// Mitsubishi GX Works2 project: 최예현_servo_exam   PLC: Q02/Q02H

PROGRAM MAIN
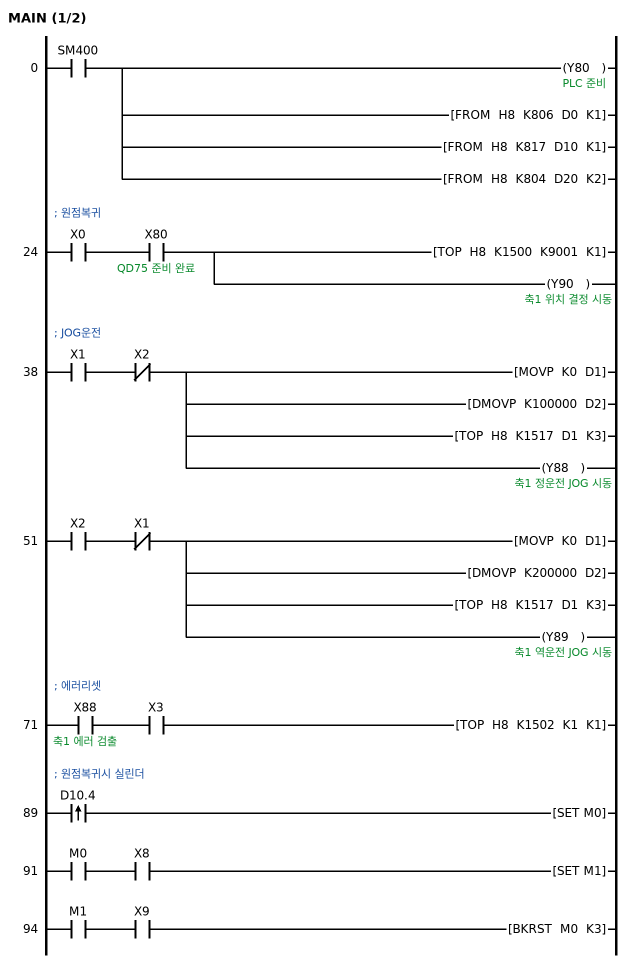
0     LD      SM400
      OUT     Y80  ; PLC 준비
      FROM    H8 K806 D0 K1
      FROM    H8 K817 D10 K1
      FROM    H8 K804 D20 K2
; 원점복귀
24    LD      X0
      AND     X80  ; QD75 준비 완료
      TOP     H8 K1500 K9001 K1
      OUT     Y90  ; 축1 위치 결정 시동
; JOG운전
38    LD      X1
      ANI     X2
      MOVP    K0 D1
      DMOVP   K100000 D2
      TOP     H8 K1517 D1 K3
      OUT     Y88  ; 축1 정운전 JOG 시동
51    LD      X2
      ANI     X1
      MOVP    K0 D1
      DMOVP   K200000 D2
      TOP     H8 K1517 D1 K3
      OUT     Y89  ; 축1 역운전 JOG 시동
; 에러리셋
71    LD      X88  ; 축1 에러 검출
      AND     X3
      TOP     H8 K1502 K1 K1
; 원점복귀시 실린더
89    LDP     D10.4
      SET     M0
91    LD      M0
      AND     X8
      SET     M1
94    LD      M1
      AND     X9
      BKRST   M0 K3
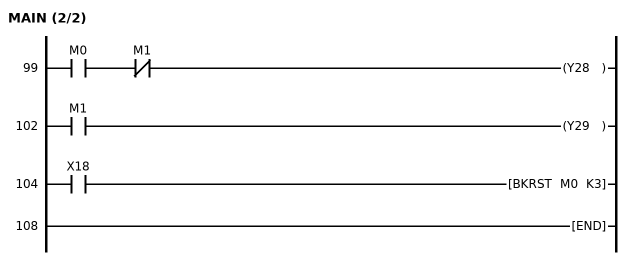
99    LD      M0
      ANI     M1
      OUT     Y28
102   LD      M1
      OUT     Y29
104   LD      X18
      BKRST   M0 K3
108   END
END_PROGRAM

// device comments not shown above
X81  ; 동기용 플래그
X84  ; 축1 M 코드 ON
X85  ; 축2 M 코드 ON
X89  ; 축2 에러 검출
X8C  ; 축1 BUSY
X8D  ; 축2 BUSY
X90  ; 축1 시동 완료
X91  ; 축2 시동 완료
X94  ; 축1 위치 결정 완료
X95  ; 축2 위치 결정 완료
Y84  ; 축1 축 정지
Y85  ; 축2 축 정지
Y8A  ; 축2 정운전 JOG 시동
Y8B  ; 축2 역운전 JOG 시동
Y91  ; 축2 위치 결정 시동
Y94  ; 축1 실행 금지 플래그
Y95  ; 축2 실행 금지 플래그
